// TIA Portal V17 export
// export: Created 2024-09-02T12:50:28.6608772Z, ExportSetting WithDefaults, DisplayName Totally Integrated Automation Portal, DisplayVersion V17, DisplayName TIA Portal Openness, DisplayVersion V17, DisplayName TIA Portal Version Control Interface, DisplayVersion V17, DisplayName STEP 7 Professional, DisplayVersion V17, DisplayName STEP 7 Safety, DisplayVersion V17, DisplayName WinCC Professional, DisplayVersion V17
TYPE "TypeSKS_MOTOR"
// stored: IsFailsafeCompliant false
   STRUCT
      "A" : Struct
         on : Bool;
         off : Bool;
         forwards : Bool;
         backwards : Bool;
         request : Bool;
         "timer" { S7_SetPoint := 'True'} : IEC_TIMER;
      END_STRUCT;
      H : Struct
         on : Bool;
         off : Bool;
         forwards : Bool;
         backwards : Bool;
      END_STRUCT;
   END_STRUCT;
END_TYPE
